FUNCTION_BLOCK FB_moveToTorque
VAR_IN_OUT
	Axis : AXIS_REF;					
END_VAR
VAR_INPUT
	Execute 			: BOOL;
	Direction 			: INT; // 0- PositiveDirection, 1- NegativeDirection
	Velocity 			: LREAL;
	Acceleration 		: LREAL;
	Deceleration 		: LREAL;
	DetectionTorqueTime : TIME;
	TorqueLimit 		: LREAL;
END_VAR
VAR_OUTPUT
	Done 			: BOOL;
	Busy 			: BOOL;
	Active 			: BOOL;
	CommandAborted 	: BOOL;
	Error 			: BOOL;
	ErrorID 		: UDINT;
END_VAR
VAR
	nState 			: INT;
	fbExecute 		: R_TRIG;
	fbDetectTime 	: TON;
	
	readParameter 		: MC_ReadParameter;
	readParameterOut 	: ST_mcOutputs;
	
	writeParameter		: MC_WriteParameter;
	writeParameterOut 	: ST_mcOutputs;
	readValue 			: LREAL;
	
	parameter 	: MC_AxisParameter;	
	writeValue 	: LREAL;
	
	moveToTorque	: MC_TorqueControl;
	torqueOptions 	: ST_TorqueControlOptions;
	moveToTorqueOut : ST_mcOutputs;
	
	moveAbsolute	: MC_MoveAbsolute;
	moveAbsoluteOut : ST_mcOutputs;
	calcBackOffPos 	: LREAL;
	
	home	: MC_Home;
	homeOut : ST_mcOutputs;
	
	stop		: MC_Stop;
	stopOut 	: ST_mcOutputs;
	fPosition	: LREAL;

	jog		: MC_Jog;
	jogOut 	: ST_mcOutputs;
	
	moveRelative	: MC_MoveRelative;
	moveRelativeOut	: ST_mcOutputs;
END_VAR

fbExecute(CLK := Execute);
fbDetectTime.PT := DetectionTorqueTime;
fbDetectTime();
actMove();


CASE nState OF 
	0: //init
		IF NOT Execute THEN
		(* reset at falling edge of Execute *)
			Busy 					:= FALSE;
			Done					:= FALSE;
			CommandAborted 			:= FALSE;
			Error 					:= FALSE;
			ErrorID 				:= 0;
			fbDetectTime.IN 		:= FALSE;
			readParameter.Enable 	:= FALSE;
			writeParameter.Execute 	:= FALSE;
			stop.Execute 			:= FALSE;
			home.Execute 			:= FALSE;
			moveAbsolute.Execute 	:= FALSE;
			jog.JogForward 			:= FALSE;
			jog.JogBackwards 		:= FALSE;
		END_IF
	
		IF fbExecute.Q THEN
			Busy := TRUE;
			nState := nState + 1;
		END_IF
		
	1: //Execute MoveTowards Torque
		CASE Direction OF
			0: //mcPositiveDirection
				jog.JogForward := TRUE;
				jog.JogBackwards := FALSE;
			1: //mcNegativeDirection
				jog.JogForward := FALSE;
				jog.JogBackwards := TRUE;
		END_CASE
			
		IF ABS(axis.NcToPlc.ActTorque) > ABS(TorqueLimit) THEN
			fbDetectTime.IN := TRUE;
			IF fbDetectTime.Q THEN
				jog.JogForward := FALSE;
				jog.JogBackwards := FALSE;
				nState := nState + 1;
			END_IF
		ELSIF NOT jogOut.Busy AND jogOut.Error THEN
			Error := jogOut.Error;
			ErrorID := jogOut.ErrorID;
			jog.JogForward := FALSE;
			jog.JogBackwards := FALSE;
			nState := 0;
		ELSIF jogOut.CommandAborted THEN
			jog.JogForward := FALSE;
			jog.JogBackwards := FALSE;
		ELSE
			fbDetectTime.IN := FALSE;
		END_IF
		
	2: // Stop motor
		stop.Execute := TRUE;
		
		IF stopOut.Busy AND stopOut.Done THEN
			stop.Execute := FALSE;
			Busy := FALSE;
			Done := TRUE;
			nState := 0;
			
		ELSIF NOT stopOut.Busy AND stopOut.Error THEN
			Error := stopOut.Error;
			ErrorId := stopOut.ErrorID;
			stop.Execute := FALSE;
			nState := 0;
		END_IF
END_CASE

IF axis.Status.Error THEN
	nState := 0;
END_IF

ACTION actMove:
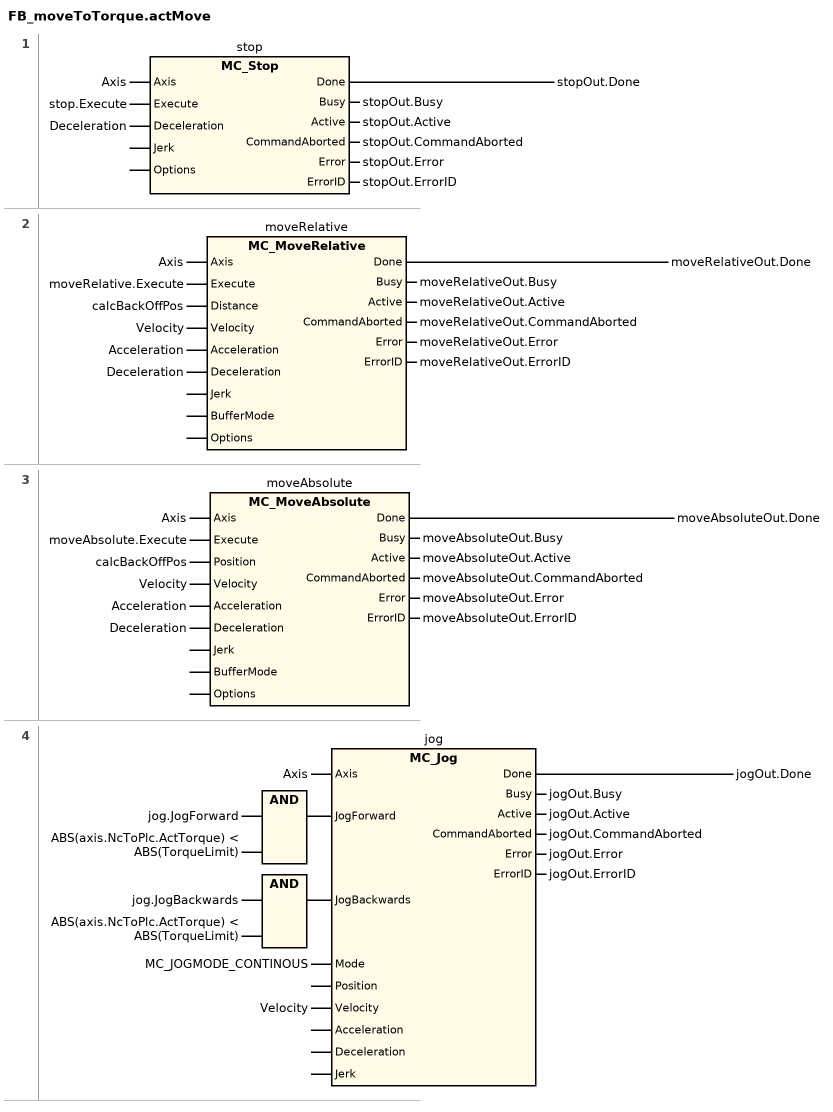
// NETWORK 1
stop(
    Axis := Axis,
    Execute := stop.Execute,
    Deceleration := Deceleration,
    Busy => stopOut.Busy,
    Active => stopOut.Active,
    CommandAborted => stopOut.CommandAborted,
    Error => stopOut.Error,
    ErrorID => stopOut.ErrorID); // MC_Stop
stopOut.Done := stop.Done;

// NETWORK 2
moveRelative(
    Axis := Axis,
    Execute := moveRelative.Execute,
    Distance := calcBackOffPos,
    Velocity := Velocity,
    Acceleration := Acceleration,
    Deceleration := Deceleration,
    Busy => moveRelativeOut.Busy,
    Active => moveRelativeOut.Active,
    CommandAborted => moveRelativeOut.CommandAborted,
    Error => moveRelativeOut.Error,
    ErrorID => moveRelativeOut.ErrorID); // MC_MoveRelative
moveRelativeOut.Done := moveRelative.Done;

// NETWORK 3
moveAbsolute(
    Axis := Axis,
    Execute := moveAbsolute.Execute,
    Position := calcBackOffPos,
    Velocity := Velocity,
    Acceleration := Acceleration,
    Deceleration := Deceleration,
    Busy => moveAbsoluteOut.Busy,
    Active => moveAbsoluteOut.Active,
    CommandAborted => moveAbsoluteOut.CommandAborted,
    Error => moveAbsoluteOut.Error,
    ErrorID => moveAbsoluteOut.ErrorID); // MC_MoveAbsolute
moveAbsoluteOut.Done := moveAbsolute.Done;

// NETWORK 4
jog(
    Axis := Axis,
    JogForward := jog.JogForward AND (ABS(axis.NcToPlc.ActTorque) < ABS(TorqueLimit)),
    JogBackwards := jog.JogBackwards AND (ABS(axis.NcToPlc.ActTorque) < ABS(TorqueLimit)),
    Mode := MC_JOGMODE_CONTINOUS,
    Velocity := Velocity,
    Busy => jogOut.Busy,
    Active => jogOut.Active,
    CommandAborted => jogOut.CommandAborted,
    Error => jogOut.Error,
    ErrorID => jogOut.ErrorID); // MC_Jog
jogOut.Done := jog.Done;
END_ACTION

END_FUNCTION_BLOCK

(* stored: Version 1.1.0.1, ProductVersion 3.1.4024.13
   POU FB_moveToTorque: Id {f0a67633-e5e7-4804-8db2-0804b85f7701}, SpecialFunc None
   Action actMove: Id {cca3905f-8572-44a5-9484-caaa85916f0d} *)
